(* Create Drive State Output *)
CASE DriveMode OF
0:
	IF bModePMActive THEN
		(* Parameterization mode active *)
		DriveState := DriveState_Mode_PM;
	ELSE
		(* Mode Invalid *)
		DriveState := DriveState_Mode_Invalid;
	END_IF
1:
	IF bModePMActive THEN
		(* Mode Invalid *)
		DriveState := DriveState_Mode_Invalid;
	ELSE
		(* 'bb' mode active *)
		DriveState := DriveState_Mode_bb;
	END_IF
2:
	IF bModePMActive THEN
		(* Mode Invalid *)
		DriveState := DriveState_Mode_Invalid;
	ELSE
		(* Ab' mode active *)
		DriveState := DriveState_Mode_Ab;
	END_IF
3:
	IF bModePMActive THEN
		(* Mode Invalid *)
		DriveState := DriveState_Mode_Invalid;
	ELSE
		IF bDriveHalt THEN
			(* 'AH' mode active *)
			DriveState := DriveState_Mode_AH;
		ELSE
			IF NOT bMLDRunning THEN
				(* 'AF' mode active *)
				DriveState := DriveState_Mode_AF;
			ELSE
				IF bPressureControlActive THEN
					(* Pressure control mode active *)
					DriveState := DriveState_Mode_PC;
				ELSE
					(* flow rate control mode active *)
					DriveState := DriveState_Mode_FC;
				END_IF
			END_IF
		END_IF
	END_IF
ELSE
	(* Mode Invalid *)
	DriveState := DriveState_Mode_Invalid;
END_CASE

(* Mode specific operations and calculations *)
CASE DriveState OF

DriveState_Mode_PC:
(* Pressure Control Mode Active *)
	CommandValueReached := bPressureCmdValReached;
	(* start Pump01 if commanded *)
	Pump01On := PumpOn;

	(* Pump02 is controlled from MLD program *)
	Pump02On := PumpOn AND bMLDPump2OnCmd;

	(* initialize total volume *)
	IF Pump01On THEN
		dwTotalVolume := VolumePump01;
		IF Pump02On THEN
			dwTotalVolume := VolumePump01 + VolumePump02;
		END_IF
	ELSE
		dwTotalVolume := 0;
	END_IF
	(* flow rate is multiplication of Act Velocity and total volume *)
	FlowrateActValue := dwTotalVolume * diVelocityAct ;
	(* transfer Pressure Command value to drive *)
	diPressureCmd := PressureCmdValue;
	(* reset velocty command *)
	diVelocityCmd := 0;

DriveState_Mode_FC:
(* Flow rate Control Mode Active *)
	(* Flow rate value reached when Velocity is within tolerance window *)
	CommandValueReached := bVelCmdValReached;
	(* start Pump01 if commanded *)
	Pump01On := PumpOn;
	(* Pump02 is on along with Pump01 *)
	Pump02On := PumpOn ;

	(* initialize total volume *)
	IF Pump01On THEN (* and Pump02 is also On *)
		dwTotalVolume := VolumePump01 + VolumePump02;
	ELSE
		dwTotalVolume := 0;
	END_IF
	(* flow rate is multiplication of Act Velocity and total volume *)
	FlowrateActValue := dwTotalVolume * diVelocityAct ;

	IF (dwTotalVolume = 0 ) THEN
		(* reset velocty command, no Volume no flow rate control *)
		diVelocityCmd := 0;
	ELSE
		(* velocty command value is derived by deviding Flowrate Command value with Total volume *)
		diVelocityCmd := FlowrateCmdValue / dwTotalVolume;
	END_IF

	(* Pressure Command zero in Flow rate control *)
	diPressureCmd := 0;
ELSE
	(* reset all outputs if not in Process Control mode *)
	dwTotalVolume := 0;
	diVelocityCmd := 0;
	FlowrateActValue := 0;
	diPressureCmd := 0;
	CommandValueReached := FALSE;
END_CASE
(* end of Mode specific operations *)

(* set Master control word and Signal control word *)
wMasterControlWord.14 := DriveEnable;
wMasterControlWord.15 := DriveStart;
wMasterControlWord.13 := DriveStart;                                       (* Drive Halt bit must be set to Activate AF mode at Drive*)

(* reset Diagnostic message using Signal control Word Bit 5 , S144 *)
wSignalControlWord.5 := ResetDriveError;

(* Command for changing the operating mode from Pressure control to Flow rate control and vice versa *)
IF ( OperatingMode = 1)  AND DriveEnable AND DriveStart THEN
	wMLDControlWord.0 := TRUE;
ELSE
	wMLDControlWord.0 := FALSE;
END_IF
(* command to open / close Pump 01 *)
wMLDControlWord.2 := Pump01On;

(* Transfer Command values to the respective output variables *)
stOutputPara.wMasterControlWord := wMasterControlWord;
fbMuxIndradrive.dwValue_WRITE_2 := WORD_TO_DWORD(wSignalControlWord);
fbMuxIndradrive.dwValue_WRITE_3 := diVelocityCmd;
fbMuxIndradrive.dwValue_WRITE_4 := diPressureCmd;
fbMuxIndradrive.dwValue_WRITE_5 := WORD_TO_DWORD (wMLDControlWord);

(*###############################################################################*)
(*####  Call Multiplex Function block and get element number '0' Read and Written Cyclically                      *)
(*###############################################################################*)
fbMuxIndradrive(
	uiINDEX_WRITE                          := OP_MODE_PROCESS_CNTRL ,
	uiLIST_INDEX_WRITE                := LIST_INDEX_0,
	dwValue_WRITE_1                     :=  ,       (* S-0-0000 - Reserve *)
	dwValue_WRITE_2                     :=  ,       (* S-0-0145 - Signal control word *)
	dwValue_WRITE_3                     :=  ,       (* S-0-0259 - Positioning Velocity*)
	dwValue_WRITE_4                     :=  ,       (* S-0-0282 - Position Command Value *)
	dwValue_WRITE_5                     :=  ,       (* S-0-0000 - Reserve *)
	dwValue_WRITE_6                     :=  ,       (* S-0-0000 - Reserve *)
	dwValue_WRITE_7                     :=  ,       (* S-0-0000 - Reserve *)
	dwValue_WRITE_8                     :=  ,       (* S-0-0000 - Reserve *)
	uiINDEX_READ                           := OP_MODE_PROCESS_CNTRL,
	uiLIST_INDEX_READ                 := LIST_INDEX_0 ,
	stEK_IN                                         := stInputPara.stMUX_in ,
	uiINDEX_WRITE_ACKNOWLEDGE=> ,
	uiLIST_INDEX_WRITE_ACKNOWLEDGE=> ,
	uiINDEX_READ_ACKNOWLEDGE=> ,
	uiLIST_INDEX_READ_ACKNOWLEDGE=> ,
	dwValue_READ_1                      => ,           (* S-0-0000 - Reserve *)
	dwValue_READ_2                      => ,           (* S-0-0144 - Signal Status word *)
	dwValue_READ_3                      => ,           (* S-0-0047 - Velocity feedback value *)
	dwValue_READ_4                      => ,           (* S-0-0051 - Postion feedback value *)
	dwValue_READ_5                      => ,           (* S-0-0390 - Drive Diagnostic word *)
	dwValue_READ_6                      => ,           (* S-0-0000 - Reserve *)
	dwValue_READ_7                      => ,           (* S-0-0000 - Reserve *)
	dwValue_READ_8                      => ,           (* S-0-0000 - Reserve *)
	stEK_OUT                                    => stOutputPara.stMUX_out);
END_FUNCTION_BLOCK

(* POU fbIndradrive, ST *)
FUNCTION_BLOCK fbIndradrive
VAR_INPUT
	In_Enable:BOOL;			(*1=Enable Drive, 0=Disable and ignore error*)
	In_Reset:BOOL;
	In_AbsEncoder:BOOL;		(*1=Absolute Encoder, 0=Incremental Encoder*)
	In_DriveInput:st_Indradrive_DCP_input ;		(*Indradrive Input Words via Ethercat*)
	In_CommState:UINT ;		(*Ethercat Slave State, 8=OK*)
	plsResetMode: R_TRIG;
END_VAR
VAR_OUTPUT
	Out_DriveOutput: st_Indradrive_DCP_output;	(*Indradrive Output Words via Ethercat*)
	Out_DriveFeedRateOverride: UINT;			(*Indradrive Output for Feedrate override, keep at 100%*)
END_VAR
VAR_IN_OUT
	DriveVar:structIndradrive;	(*Local Data structure to handle Indradrive variables*)
	Station:Struc_Station_Ctrl ;
END_VAR
VAR
	Drive: FB_Indradrive_DCP;	(*Standard Function Block Provided by Bosch*)
	tmrDriveEnableTOUT:TON;
	tmrHomingTOUT:TON;
	tmrMovePosTOUT:TON;
	diPosCmd:DINT;
	diVelCmd:DINT;
	DriveStatus:INT;
	plsInPos: R_TRIG;
	plsLimitTriggered: R_trig;
	plsMoveRel: R_trig;
	plsStopMove: R_TRIG;
	plsEMGReset: R_trig;
	ServoBusy:BOOL;
	NotAbsEncHoming:BOOL;
	plsMoveAbs: R_trig;
	plsStopMove2: R_trig;
END_VAR
VAR CONSTANT
	FACTOR_DINT_REAL : INT := 10000;
	FACTOR_VEL_DINT_REAL : INT := 1000;
END_VAR
(* convert DINT values from FB to REAL values for the user program and vise versa*)
(* used only for trace purpose *)
DriveVar.Out_CurrPos := DINT_TO_REAL(Drive.diPOS_ACT) / FACTOR_DINT_REAL;
DriveVar.Out_CurrVel := DINT_TO_REAL(Drive.diVEL_ACT) / FACTOR_VEL_DINT_REAL;

(* REAL variables can be used for commanding instead of DINT variable used in the sample code *)
Drive.diPOS_CMD := REAL_TO_DINT (DriveVar.In_PosCmd * FACTOR_DINT_REAL);
Drive.diVEL_CMD := REAL_TO_DINT (DriveVar.In_VelCmd * FACTOR_VEL_DINT_REAL);

(*Force Slow Speed in Manual Mode When close to Negative Limit For Accurate Referencing*)
IF DriveVar.Out_CurrPos <= 20 AND DriveVar.In_JogBwd THEN
	Drive.diVEL_CMD := 60 * FACTOR_VEL_DINT_REAL;
END_IF

IF mc.ManualMode AND DriveVar.In_VelCmd > 1000 THEN
	DriveVar.In_VelCmd := 1000;
END_IF

Out_DriveFeedRateOverride := 100;

(***********************************************************************************************)
(*Servo Controller Status*)

IF NOT In_DriveInput.wSignalstatuswort.11 AND NOT In_DriveInput.wSignalstatuswort.12 THEN
	DriveStatus := 0;	(* Control section and power section not ready for operation (e.g., drive error or phase 2)*)
ELSIF NOT In_DriveInput.wSignalstatuswort.11 AND In_DriveInput.wSignalstatuswort.12 THEN
	DriveStatus := 1;	(* Control section ready for operation (bb)*)
ELSIF In_DriveInput.wSignalstatuswort.11 AND NOT In_DriveInput.wSignalstatuswort.12 THEN
	DriveStatus := 2;	(* Control section and power section ready for operation (Ab)*)
ELSIF In_DriveInput.wSignalstatuswort.11 AND In_DriveInput.wSignalstatuswort.12 THEN
	DriveStatus := 3;	(* Drive with torque (AF)*)
END_IF

(***********************************************************************************************)
(*Servo Limit Sensors Status*)
DriveVar.Out_PosLimit := In_DriveInput.wSignalstatuswort.13;
DriveVar.Out_NegLimit := In_DriveInput.wSignalstatuswort.14;

(***********************************************************************************************)
(*Error Handling*)

IF In_Reset THEN
	DriveVar.Out_ErrorWord := 0;
END_IF

Drive.bRESET := In_Reset;

(*Servo is in Alarm State Error*)
IF Drive.bERROR AND In_Enable  THEN
	DriveVar.Out_ErrorWord := 11;
END_IF

(*Servo Control and Power Section Not Ready Error*) 
IF DriveStatus = 0 AND In_Enable  THEN
	DriveVar.Out_ErrorWord := 12;
END_IF

(*Servo Enable Timeout Error*) 
tmrDriveEnableTOUT(IN:= Drive.bDRIVE_ENABLE AND NOT (Drive.bQ_DRIVE_ENABLE ),PT:=T#5S);
IF tmrDriveEnableTOUT.Q AND In_Enable THEN
	DriveVar.Out_ErrorWord := 13;
END_IF

(*Servo Not Referenced Error*)
IF Drive.bQ_DRIVE_ENABLE AND NOT Drive.bIN_REFERENCE AND In_AbsEncoder AND In_Enable  THEN
	DriveVar.Out_ErrorWord := 20;
END_IF

(*Servo Homing Timeout Error*) 
tmrHomingTOUT(IN:= Drive.bHOMING,PT:=T#3000S);
IF tmrHomingTOUT.Q THEN 
	DriveVar.Out_ErrorWord := 21;
	Drive.bHOMING := FALSE;
END_IF

(*Servo Move Position Timeout Error*) 
tmrMovePosTOUT(IN:= (DriveVar.In_MoveAbs OR ServoBusy OR
					DriveVar.In_MoveRel) AND NOT DriveVar.Out_InPos,PT:=T#300S);
IF tmrMovePosTOUT.Q THEN 
	DriveVar.Out_ErrorWord := 22;
	ServoBusy := FALSE;
	DriveVar.In_MoveAbs := FALSE;
	DriveVar.In_MoveRel := FALSE;
END_IF

(*Servo Move Position Limit Error*) 
IF ServoBusy AND
	(((DriveVar.In_PosCmd < DriveVar.Out_CurrPos) AND NOT DriveVar.Out_NegLimit) 
	OR ((DriveVar.In_PosCmd > DriveVar.Out_CurrPos) AND NOT DriveVar.Out_PosLimit)) THEN 
	DriveVar.Out_ErrorWord := 23;
	ServoBusy := FALSE;
	DriveVar.In_MoveAbs := FALSE;
	DriveVar.In_MoveRel := FALSE;
END_IF

(*Servo Communication Error*) 
IF In_CommState <> 8 AND In_Enable  THEN
	DriveVar.Out_ErrorWord := 10;
END_IF

IF DriveVar.Out_ErrorWord > 1 THEN
	DriveVar.Out_Error := TRUE;
ELSE
	IF NOT DriveVar.In_MoveXLock THEN
		DriveVar.Out_ErrorWord := 0;
	ELSE
		DriveVar.Out_ErrorWord := 1;
	END_IF
	DriveVar.Out_Error := FALSE;
END_IF
(*Warning*)
DriveVar.Out_Warning := Drive.bWARNING;

(***********************************************************************************************)
(*Servo Enable*)

plsLimitTriggered(CLK:=NOT (DriveVar.Out_NegLimit AND DriveVar.Out_PosLimit) AND NOT NotAbsEncHoming);

IF plsLimitTriggered.Q THEN
	DriveVar.In_ServoOn		 := FALSE;
END_IF

IF In_Enable AND DriveVar.In_ServoOn AND NOT DriveVar.Out_Error
	AND DriveStatus >= 1  THEN
	(* drive enable and drive on commands *)
	Drive.bDRIVE_ENABLE	:= TRUE;
	Drive.bDRIVE_START		:= TRUE;
ELSE
	(* drive enable and drive on commands *)
	Drive.bDRIVE_ENABLE	:= FALSE;
	Drive.bDRIVE_START		:= FALSE;
	DriveVar.Out_Busy 		:= FALSE;
	DriveVar.In_JogBwd 		:= FALSE;
	DriveVar.In_JogFwd 		:= FALSE;
	DriveVar.In_MoveAbs 		:= FALSE;
	DriveVar.In_MoveHome 	:= FALSE;
	DriveVar.In_MoveRel 		:= FALSE;
	DriveVar.In_ServoOn 		:= FALSE;
END_IF

Drive.bIMMEDIATE_CHANGE := TRUE;
	
(***********************************************************************************************)
(*Servo Movement Control*)
(***********************************************************************************************)

(*Force Stop Command When Mode Changes*)
plsResetMode(CLK:= NOT MC.AutoMode);

plsStopMove(CLK:= NOT (Station.OriginSchRun OR MC.OriginSchRun OR
						Station.AutoRun OR Station.M_Step));

plsStopMove2(CLK:= (Station.OriginSchRun OR MC.OriginSchRun OR
						Station.M_Step OR MC.AutoMode));
						
IF plsStopMove.Q AND plsStopMove2.Q OR plsResetMode.Q THEN
	DriveVar.In_StopMove := TRUE;
	DriveVar.In_MoveAbs := FALSE;
	DriveVar.In_MoveHome := FALSE;
	DriveVar.In_MoveRel := FALSE;
END_IF

(*Check New Move Command Direction for Interlocking Purpose*)
IF DriveVar.In_JogFwd OR 
	((DriveVar.In_PosCmd > DriveVar.Out_CurrPos) AND
		DriveVar.In_MoveAbs) OR
	((DriveVar.In_PosCmd > 0) AND
		DriveVar.In_MoveRel) THEN
	DriveVar.Out_PosDirc := TRUE;
	DriveVar.Out_NegDirc := FALSE;
ELSIF DriveVar.In_JogBwd OR 
	((DriveVar.In_PosCmd < DriveVar.Out_CurrPos) AND
		DriveVar.In_MoveAbs) OR
	((DriveVar.In_PosCmd < 0) AND
		DriveVar.In_MoveRel) THEN	
	DriveVar.Out_PosDirc := FALSE;
	DriveVar.Out_NegDirc := TRUE;
ELSE
	DriveVar.Out_PosDirc := FALSE;
	DriveVar.Out_NegDirc := FALSE;
END_IF


(* Origin Search for Incremental Encoder Servo*)
	IF NOT In_AbsEncoder THEN
		IF Drive.bIN_REFERENCE OR NOT DriveVar.In_ServoOn THEN
			Drive.bHOMING 		:= FALSE;
			NotAbsEncHoming	:=FALSE;
		END_IF

		IF DriveVar.In_MoveHome  AND
			Drive.bQ_DRIVE_ENABLE AND
			DriveStatus = 3  AND
			NOT DriveVar.Out_Busy THEN
			Drive.bHOMING 		:= TRUE;
			NotAbsEncHoming	:=TRUE;
		END_IF
	END_IF

IF Drive.bQ_DRIVE_ENABLE AND Drive.bQ_MAIN_MODE AND DriveStatus = 3 THEN
	DriveVar.Out_Ready := TRUE;
	


	(*Jog Command*)
	IF MC.ManualMode AND NOT Station.M_Step THEN
		IF DriveVar.In_JogFwd AND NOT DriveVar.In_JogBwd AND DriveVar.In_MoveXLock THEN
			(* Jog Positive command *)
			Drive.bJOG_FORWARD := TRUE;
			Drive.bJOG_BACKWARD := FALSE;
		ELSIF NOT DriveVar.In_JogFwd AND DriveVar.In_JogBwd AND DriveVar.In_MoveXLock THEN
			(* Jog Negative  command *)
			Drive.bJOG_FORWARD := FALSE;
			Drive.bJOG_BACKWARD := TRUE;
		ELSE
			(* Stop Jogging *)
			Drive.bJOG_FORWARD := FALSE;
			Drive.bJOG_BACKWARD := FALSE;
		END_IF
	ELSE
		DriveVar.In_JogFwd := FALSE;
		DriveVar.In_JogBwd := FALSE;
	END_IF
	
	IF Drive.bIN_REFERENCE THEN
		IF DriveVar.In_MoveXLock THEN
			(* Start Absolute move *)
			plsMoveAbs(CLK:=DriveVar.In_MoveAbs);
			IF DriveVar.In_MoveAbs AND Drive.bNEW_VALUE_POSSIBLE THEN
				ServoBusy := TRUE;
				(*DriveVar.In_MoveAbs := FALSE;*)
				IF Drive.diPOS_CMD <> Drive.diPOS_ACT AND Drive.diVEL_CMD <> 0 THEN
					DriveVar.Out_InPos := FALSE;
					Drive.bABS_REL := FALSE;       				(* False --> Absolute command *)
					IF Drive.bNEW_VALUE THEN
						Drive.bNEW_VALUE := FALSE;
					ELSE
						Drive.bNEW_VALUE := TRUE;
					END_IF
				END_IF
			END_IF
			(* Start Relative move *)
			plsMoveRel(CLK:=DriveVar.In_MoveRel);
			IF plsMoveRel.Q AND Drive.bNEW_VALUE_POSSIBLE AND 
				NOT ServoBusy  THEN
				ServoBusy := TRUE;
				DriveVar.In_MoveRel := FALSE;
				IF Drive.diPOS_CMD <> 0 AND Drive.diVEL_CMD <> 0 THEN
					DriveVar.Out_InPos := FALSE;
					Drive.bABS_REL := TRUE;       				(* True  --> Relative  command *)
					IF Drive.bNEW_VALUE THEN
						Drive.bNEW_VALUE := FALSE;
					ELSE
						Drive.bNEW_VALUE := TRUE;
					END_IF
				END_IF
			END_IF
		END_IF
	ELSE
		DriveVar.Out_InPos := FALSE;
	END_IF
	
	(*Set Servo Busy Status*)	
	DriveVar.Out_Busy := NOT Drive.bIN_STANDSTILL;
	IF DriveVar.Out_Busy THEN
		DriveVar.Out_InPos := FALSE; 
	END_IF
	
ELSE

	ServoBusy 				:= FALSE;
	DriveVar.In_MoveAbs 		:= FALSE;
	DriveVar.In_MoveRel		 := FALSE;
	DriveVar.Out_Ready		:= FALSE;
	DriveVar.In_JogBwd		 := FALSE;
	DriveVar.In_JogFwd 		:= FALSE;
(*	DriveVar.In_MoveHome 	:= FALSE;*)
	Drive.bJOG_FORWARD	:= FALSE;
	Drive.bJOG_BACKWARD	 := FALSE;
	Drive.bHOMING			 := FALSE;

END_IF

(* wait for InPos *)
plsInPos(CLK:= Drive.bPOS_OK);
plsEMGReset(CLK:= NOT MC.Trouble );
IF Drive.bPOS_OK AND 
	fcComparePos(CurrPos:= DriveVar.In_PosCmd, TargetPos:= DriveVar.Out_CurrPos,Tolerance:=0.5)
	AND Drive.bIN_STANDSTILL AND Drive.bNEW_VALUE_POSSIBLE  THEN
	DriveVar.Out_InPos 		:= TRUE;
	DriveVar.In_MoveAbs 		:= FALSE;
	DriveVar.In_MoveRel		:= FALSE;
	ServoBusy 				:= FALSE;
END_IF

IF plsEMGReset.Q AND Drive.bIN_STANDSTILL AND Drive.bIN_REFERENCE AND
	Drive.bNEW_VALUE_POSSIBLE THEN
	DriveVar.Out_InPos		:= TRUE;
	ServoBusy 				:= FALSE;
END_IF

IF DriveVar.In_StopMove THEN
	DriveVar.In_MoveAbs 		:= FALSE;
	DriveVar.In_MoveHome	:= FALSE;
	DriveVar.In_MoveRel		:= FALSE;
	DriveVar.In_JogBwd 		:= FALSE;
	DriveVar.In_JogFwd		:= FALSE;
	DriveVar.In_StopMove 		:= FALSE;
	(* Stop Movement *)
	Drive.bJOG_FORWARD	:= TRUE;
	Drive.bJOG_BACKWARD 	:= TRUE;
	ServoBusy 				:= FALSE;

ELSIF 	Drive.bJOG_FORWARD AND Drive.bJOG_BACKWARD AND MC.AutoMode THEN
	Drive.bJOG_FORWARD 	:= FALSE;
	Drive.bJOG_BACKWARD 	:= FALSE;
END_IF


(***********************************************************************************************)
(*Servo Function Block*)


Drive(
	bJOG_FORWARD:= 			,
	bJOG_BACKWARD:=			,
	bNEW_VALUE:= ,
	bABS_REL:= ,
	bIMMEDIATE_CHANGE:= ,
	diPOS_CMD:= ,
	diVEL_CMD:= , 
	stEK_IN:=					In_DriveInput ,
	bQ_DRIVE_ENABLE=> ,
	bQ_MAIN_MODE=> , 
	bIN_REFERENCE=> , 
	bPOS_OK=> , 
	bNEW_VALUE_POSSIBLE=> , 
	bSTATUS_MESSAGE=> , 
	bWARNING=> , 
	bERROR=> , 
	bIN_STANDSTILL=> , 
	dwDRIVE_DIAGNOSIS=> , 
	diPOS_ACT=> , 
	diVEL_ACT=> ,
	stEK_OUT=>					Out_DriveOutput );


	Out_DriveOutput.wSignalsteuerwort.6 	:= drive.bJOG_FORWARD;
	Out_DriveOutput.wSignalsteuerwort.7 	:= drive.bJOG_BACKWARD;
	Out_DriveOutput.wSignalsteuerwort.15 :=  NotAbsEncHoming  ;

	
(***********************************************************************************************)
(*Set Reference Point for Absulute Encoder Servo*)
	Out_DriveOutput.wSignalsteuerwort.1 := DriveVar.In_SetAbsRef;
	DriveVar.Out_Referenced := Drive.bIN_REFERENCE;
END_FUNCTION_BLOCK

(* POU fcComparePos, ST *)
FUNCTION fcComparePos : BOOL
VAR_INPUT
	CurrPos		:REAL;
	TargetPos	:REAL;
	Tolerance	:REAL;
END_VAR
VAR
END_VAR
IF 	CurrPos >= 	(TargetPos	-	Tolerance) AND
	CurrPos <= 	(TargetPos	+	Tolerance) THEN
	fcComparePos := TRUE;
ELSE
	fcComparePos := FALSE;
END_IF
END_FUNCTION

(* POU Std_Cylinder_Ctrl, LD *)
FUNCTION_BLOCK Std_Cylinder_Ctrl

VAR_INPUT
	IN:BOOL;
	IN_CylName:STRING;
	In_Enable:BOOL;
	In_Reset:BOOL;


	(*Trigger*)
	In_AutoWork:BOOL;
	In_AutoHome:BOOL;
	In_OrgWork:BOOL;
	In_OrgHome:BOOL;
	(*Mechanical Interlock*)
	In_WorkXLock:BOOL;
	In_HomeXLock:BOOL;
	(*Sensors*)
	In_WorkRS:BOOL;
	In_HomeRS:BOOL;

	(*Timer*)
	In_WorkTON:TIME;
	In_HomeTON:TIME;
	in_Timeout:TIME;
END_VAR

VAR_OUTPUT
	Q:BOOL;
	Out_WorkSV:BOOL;
	Out_HomeSV:BOOL;
	E_WorkErr:BOOL;
	E_HomeErr:BOOL;
	S_WorkPos:BOOL;
	S_HomePos:BOOL;
END_VAR

VAR
	(* Trigger*)
	T_ManWork:BOOL;
	T_ManHome:BOOL;

	Loc_Work:BOOL;
	Loc_Home:BOOL;
	Err_Cyl:BOOL;
	Fwd_TOut: TON;
	Bwd_TOut: TON;
	Fwd_TON: TON;
	Bwd_TON: TON;
	Loc_WorkPls: BOOL;
	FwdPls: R_TRIG;
	BwdPls: R_TRIG;
	Loc_HomePls: BOOL;
	Out_RSErr:BOOL;
	FwdPosPls: F_TRIG;
	BwdPosPls: F_TRIG;
END_VAR
VAR_IN_OUT

END_VAR
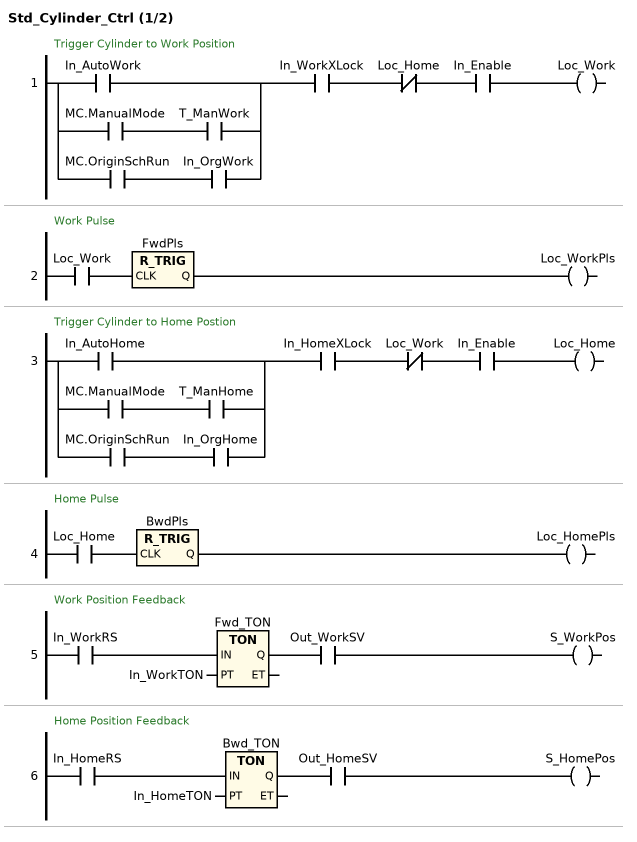
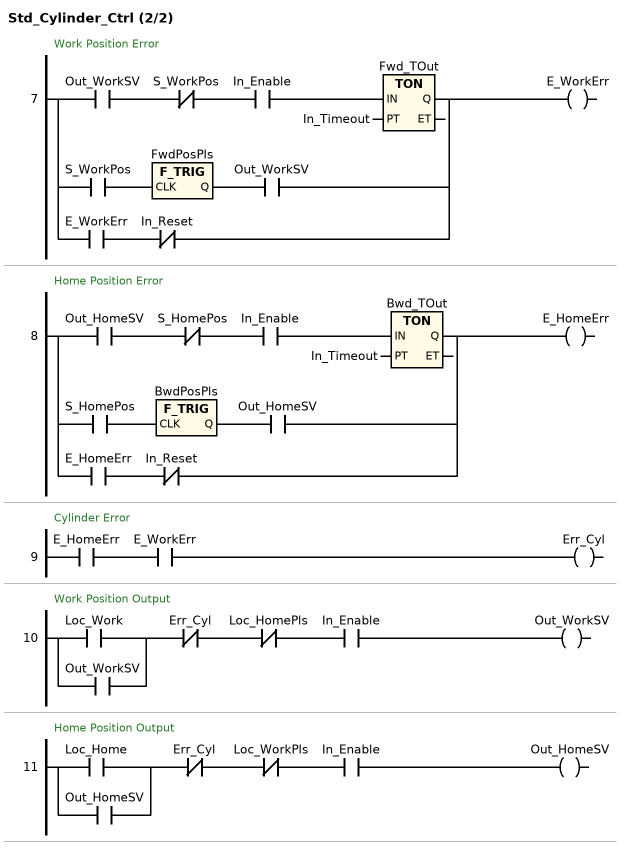
_LD_ (* Ladder Diagram *)
NETWORK 1 (* Trigger Cylinder to Work Position *)
	{ [In_AutoWork] | [MC.ManualMode] - [T_ManWork] | [MC.OriginSchRun] - [In_OrgWork] } - [In_WorkXLock] - [/Loc_Home] - [In_Enable] --- (Loc_Work)
NETWORK 2 (* Work Pulse *)
	[Loc_Work] - FwdPls:R_TRIG(CLK: *) --- (Loc_WorkPls)
NETWORK 3 (* Trigger Cylinder to Home Postion *)
	{ [In_AutoHome] | [MC.ManualMode] - [T_ManHome] | [MC.OriginSchRun] - [In_OrgHome] } - [In_HomeXLock] - [/Loc_Work] - [In_Enable] --- (Loc_Home)
NETWORK 4 (* Home Pulse *)
	[Loc_Home] - BwdPls:R_TRIG(CLK: *) --- (Loc_HomePls)
NETWORK 5 (* Work Position Feedback *)
	[In_WorkRS] - Fwd_TON:TON(IN: *, PT: In_WorkTON) - [Out_WorkSV] --- (S_WorkPos)
NETWORK 6 (* Home Position Feedback *)
	[In_HomeRS] - Bwd_TON:TON(IN: *, PT: In_HomeTON) - [Out_HomeSV] --- (S_HomePos)
NETWORK 7 (* Work Position Error *)
	{ [Out_WorkSV] - [/S_WorkPos] - [In_Enable] - Fwd_TOut:TON(IN: *, PT: In_Timeout) | [S_WorkPos] - FwdPosPls:F_TRIG(CLK: *) - [Out_WorkSV] | [E_WorkErr] - [/In_Reset] } --- (E_WorkErr)
NETWORK 8 (* Home Position Error *)
	{ [Out_HomeSV] - [/S_HomePos] - [In_Enable] - Bwd_TOut:TON(IN: *, PT: In_Timeout) | [S_HomePos] - BwdPosPls:F_TRIG(CLK: *) - [Out_HomeSV] | [E_HomeErr] - [/In_Reset] } --- (E_HomeErr)
NETWORK 9 (* Cylinder Error *)
	[E_HomeErr] - [E_WorkErr] --- (Err_Cyl)
NETWORK 10 (* Work Position Output *)
	{ [Loc_Work] | [Out_WorkSV] } - [/Err_Cyl] - [/Loc_HomePls] - [In_Enable] --- (Out_WorkSV)
NETWORK 11 (* Home Position Output *)
	{ [Loc_Home] | [Out_HomeSV] } - [/Err_Cyl] - [/Loc_WorkPls] - [In_Enable] --- (Out_HomeSV)
_END_LD_
(* the same logic as Structured Text *)
(* Network 1: Trigger Cylinder to Work Position *)
Loc_Work := (In_AutoWork OR MC.ManualMode AND T_ManWork OR MC.OriginSchRun AND In_OrgWork) AND In_WorkXLock AND NOT Loc_Home AND In_Enable;
(* Network 2: Work Pulse *)
FwdPls(CLK := Loc_Work);
Loc_WorkPls := FwdPls.Q;
(* Network 3: Trigger Cylinder to Home Postion *)
Loc_Home := (In_AutoHome OR MC.ManualMode AND T_ManHome OR MC.OriginSchRun AND In_OrgHome) AND In_HomeXLock AND NOT Loc_Work AND In_Enable;
(* Network 4: Home Pulse *)
BwdPls(CLK := Loc_Home);
Loc_HomePls := BwdPls.Q;
(* Network 5: Work Position Feedback *)
Fwd_TON(IN := In_WorkRS, PT := In_WorkTON);
S_WorkPos := Fwd_TON.Q AND Out_WorkSV;
(* Network 6: Home Position Feedback *)
Bwd_TON(IN := In_HomeRS, PT := In_HomeTON);
S_HomePos := Bwd_TON.Q AND Out_HomeSV;
(* Network 7: Work Position Error *)
Fwd_TOut(IN := Out_WorkSV AND NOT S_WorkPos AND In_Enable, PT := In_Timeout);
FwdPosPls(CLK := S_WorkPos);
E_WorkErr := Fwd_TOut.Q OR FwdPosPls.Q AND Out_WorkSV OR E_WorkErr AND NOT In_Reset;
(* Network 8: Home Position Error *)
Bwd_TOut(IN := Out_HomeSV AND NOT S_HomePos AND In_Enable, PT := In_Timeout);
BwdPosPls(CLK := S_HomePos);
E_HomeErr := Bwd_TOut.Q OR BwdPosPls.Q AND Out_HomeSV OR E_HomeErr AND NOT In_Reset;
(* Network 9: Cylinder Error *)
Err_Cyl := E_HomeErr AND E_WorkErr;
(* Network 10: Work Position Output *)
Out_WorkSV := (Loc_Work OR Out_WorkSV) AND NOT Err_Cyl AND NOT Loc_HomePls AND In_Enable;
(* Network 11: Home Position Output *)
Out_HomeSV := (Loc_Home OR Out_HomeSV) AND NOT Err_Cyl AND NOT Loc_WorkPls AND In_Enable;
END_FUNCTION_BLOCK

(* POU Std_Hist_StepCase, ST *)
FUNCTION_BLOCK Std_Hist_StepCase

VAR_INPUT
	IN:BOOL;
	CurrentStep:INT;
	NextStep:INT;
END_VAR

VAR_OUTPUT
	Q:BOOL;
	NewStep:INT;
END_VAR

VAR
	StepData:ARRAY[0..100] OF Struc_Hist_Step_Case ;

	StepTimer: TON;
	Loop: INT;
END_VAR
IF CurrentStep = NextStep THEN
StepTimer(IN:=TRUE , PT:=t#1100h , Q=> , ET=> );

StepData[0].CurrentStepHist :=CurrentStep;

ELSE
(* Copy HIstory File *)
FOR Loop := 0 TO 99 DO
StepData[100-Loop].CurrentStepHist   := StepData[99-Loop].CurrentStepHist ;
StepData[100-Loop].NextStepHist := StepData[99-Loop].NextStepHist ;
StepData[100-Loop].StepTime := StepData[99-Loop].StepTime;
END_FOR

(* Update New Data*)
StepData[1].NextStepHist:=NextStep;
StepData[1].StepTime :=StepTimer.ET;

StepTimer(IN:=FALSE , PT:=T#1100h , Q=> , ET=> );
NewStep:=NextStep;
END_IF
END_FUNCTION_BLOCK

(* POU Std_IAI_16Point, ST *)
(* @OBJECTFLAGS := '0, 8' *)
FUNCTION_BLOCK Std_IAI_16Point
VAR_INPUT
	In_Enable:BOOL;
	In_Name:STRING;
	In_AutoMode:BOOL;

	(*Trigger*)
	In_AutoStart:BOOL;
	In_OrgHome:BOOL;

	In_Pos_Num:WORD;
	In_ALM:BOOL;
	In_Reset:BOOL;
	In_PEND:BOOL;
	In_HEND:BOOL;
	In_Mec_Interlock:BOOL;
	In_PosTON:TIME;
	In_Timeout:TIME;
END_VAR

VAR_OUTPUT
	S_InPos:BOOL;  (*Current Pos*)
	S_Pos_Num : INT;
	S_InHome:BOOL;
	Out_CSTR:BOOL;
	Out_PC1:BOOL;
	Out_PC2:BOOL;
	Out_PC4:BOOL;
	Out_PC8:BOOL;
	E_Alm:BOOL;
	E_AlmPos:BOOL;
END_VAR

VAR
	(* Trigger*)
	T_ManStart:BOOL;
	T_ManHome:BOOL;
	T_ManPos_Num:INT;

	CSTR:BOOL; (*Common Start Bit*)
	Home : BOOL;
	Pos_Num:INT;

	TimePos: TON;
	BitPos1: BOOL;
	BitPos2: BOOL;
	BitPos3: BOOL;
	BitPos4: BOOL;
	TimeOut: TON;
	TempBit1: BYTE;
	TempBit2: BYTE;
	TempBit3: BYTE;
	TempBit4: BYTE;
	BytePos: BYTE;
	IAI_TimeOut: BOOL;
	Error_Alm: BOOL;
	DoneTon: BOOL;
	tmrStartDelay: TON;
	StartDelayTon: BOOL;
	plsStart: R_TRIG;
	StartDelayPls: BOOL;
	plsIAIDone: R_TRIG;
	DonePls: BOOL;
	plsHome: R_TRIG;
	HomePls: BOOL;
	HomeSearch: BOOL;
	test: BOOL;
	test1: BOOL;
	tmrStartDelay_1: TON;
	StartDelayTon_1: BOOL;
	IAI_Busy: BOOL;
	test_1: BOOL;
	tmrStartDelay_Home: TON;
	StartDelayTon_Home: BOOL;
	tmrStartDelay_Home_1: TON;
	StartDelayTon_Home_1: BOOL;
END_VAR
(**************************************************************************************************************)
(*Trigger*)
(**************************************************************************************************************)
IF  In_AutoStart OR (MC.ManualMode AND T_ManStart) THEN
CSTR := TRUE;
ELSE
CSTR := FALSE;
END_IF;

IF In_AutoMode THEN
Pos_Num := In_Pos_Num;
ELSE
Pos_Num:=T_ManPos_Num;
END_IF


IF (MC.OriginSchRun AND In_OrgHome) OR (MC.ManualMode AND T_ManHome) THEN
Home := TRUE;
Pos_Num:=0;
ELSE
Home := FALSE;
END_IF;
(**************************************************************************************************************)
(*Reset Error/Warning*)
(**************************************************************************************************************)
IF In_reset AND ( E_AlmPos OR E_Alm OR Error_Alm) THEN
	E_AlmPos :=FALSE;
	E_Alm:= FALSE;
	Error_Alm := FALSE;
END_IF;

(**************************************************************************************************************)
(*System Error*)
(**************************************************************************************************************)
(* Time Out*)
TimeOut (IN := Out_CSTR AND NOT S_InPos AND  In_Mec_Interlock, PT:=In_Timeout);
IAI_TimeOut := TimeOut.Q;

IF IAI_TimeOut AND In_Enable THEN
	E_AlmPos := TRUE;
END_IF;

(* IAI Controller Error*)
IF In_Enable AND In_ALM THEN
	E_Alm := TRUE;
END_IF;

(* IAI System In Error Condition*)
Error_Alm := E_AlmPos OR E_Alm;

IF Error_Alm THEN
	Out_CSTR := FALSE;
	S_InPos := FALSE;
	HomeSearch := FALSE;
	IAI_Busy:= FALSE;
END_IF;

(**************************************************************************************************************)
(*Moving To Target Position*)
(**************************************************************************************************************)

Out_PC1 := FALSE;
Out_PC2 := FALSE;
Out_PC4 := FALSE;
Out_PC8 := FALSE;

IF In_Enable AND NOT Error_Alm THEN
	BytePos := INT_TO_BYTE (Pos_Num);
	TempBit1 := BytePos AND 2#1;
	TempBit2 := BytePos AND 2#10;
	TempBit3 := BytePos AND 2#100;
	TempBit4 := BytePos AND 2#1000;

	BitPos1 := INT_TO_BOOL (TempBit1);
	BitPos2 := INT_TO_BOOL (TempBit2);
	BitPos3 := INT_TO_BOOL (TempBit3);
	BitPos4 := INT_TO_BOOL (TempBit4);

		IF BitPos1 THEN
			Out_PC1 := TRUE;
		END_IF;

		IF BitPos2 THEN
			Out_PC2 := TRUE;
		END_IF;

		IF BitPos3 THEN
			Out_PC4 := TRUE;
		END_IF;

		IF BitPos4 THEN
			Out_PC8 := TRUE;
		END_IF;
END_IF;

(**************************************************************************************************************)
(*Moving To Target Position Common*)
(**************************************************************************************************************)
tmrStartDelay(IN := CSTR , PT:= T#0.1s);
StartDelayTon := tmrStartDelay.Q;

plsStart(CLK := StartDelayTon);
StartDelayPls := plsStart.Q;

tmrStartDelay_1(IN := Out_CSTR , PT:= T#0.5s);
StartDelayTon_1 := tmrStartDelay_1.Q;

IF In_Enable AND NOT HomeSearch AND In_Mec_Interlock AND NOT Error_Alm THEN
	IF  StartDelayPls AND In_PEND THEN
		Out_CSTR := TRUE;
		S_InPos := FALSE;
		IAI_Busy := TRUE;
	END_IF;

	IF (StartDelayTon_1 AND Out_CSTR) OR NOT In_PEND  THEN
		Out_CSTR := FALSE;
	END_IF;
END_IF;

(**************************************************************************************************************)
(*Moving Done Complete Status*)
(**************************************************************************************************************)

TimePos (IN :=  In_PEND  AND (IAI_Busy OR HomeSearch) , PT:= In_PosTON);
DoneTon := TimePos.Q;

plsIAIDone(CLK := DoneTon);
DonePls := plsIAIDone.Q;

IF DoneTon AND In_Enable THEN
	IF HomeSearch THEN
		S_Pos_Num := 0;
	ELSE
		S_Pos_Num := Pos_Num;
	END_IF
	S_InPos := TRUE;
	HomeSearch := FALSE;
	IAI_Busy:= FALSE;
END_IF;

(**************************************************************************************************************)
(*Moving Target To Home = Pos 0*)
(**************************************************************************************************************)
S_InHome := S_Pos_Num = 0 AND S_InPos AND In_HEND;

tmrStartDelay_Home(IN := Home   , PT:= T#0.1s);
StartDelayTon_Home := tmrStartDelay_Home.Q;

plsHome (CLK:= StartDelayTon_Home AND NOT IAI_Busy );
HomePls:= plsHome.Q;

tmrStartDelay_Home_1(IN := HomeSearch AND Out_CSTR , PT:= T#0.5s);
StartDelayTon_Home_1 := tmrStartDelay_Home_1.Q;

IF In_Enable AND NOT Error_Alm AND In_Mec_Interlock AND  NOT Out_CSTR  THEN
	IF HomePls THEN
		HomeSearch := TRUE;
		Out_CSTR :=TRUE;
	END_IF;
END_IF;

IF HomeSearch AND StartDelayTon_Home_1 THEN
	Out_CSTR := FALSE;
END_IF;
END_FUNCTION_BLOCK

(* POU Std_IV_Vision_Ctrl, LD *)
FUNCTION_BLOCK Std_IV_Vision_Ctrl
VAR_INPUT
	IN: BOOL;
	In_Name:STRING;
	In_Enable:BOOL;
	In_Alm:BOOL;
	In_Reset:BOOL;
	In_AutoMode:BOOL;
	In_Auto_Model:INT;
	In_Busy:BOOL;
	In_AutoTrigger:BOOL;
	In_Result:BOOL;
	In_Timeout:TIME;
END_VAR

VAR_OUTPUT
	Q:BOOL;
	Out_ProgBit0:BOOL;
	Out_ProgBit1:BOOL;
	Out_ProgBit2:BOOL;
	Out_ProgBit3:BOOL;
	Out_Trigger:BOOL;
	Out_ClearErr:BOOL;
	S_Result:BOOL;
	S_Done:BOOL;
	E_Alm:BOOL;
END_VAR

VAR
	T_ManualTrigger:	BOOL;
	T_Manual_Model:	INT;
	Model:			INT;
	Start:			BOOL;

	TempModel: BYTE;
	ModelBit1: BYTE;
	ModelBit2: BYTE;
	ModelBit3: BYTE;
	ModelBit0: BYTE;
	TimeOut: TON;
	Reset_Result: BOOL;
	Vision_Trigger: R_TRIG;
	tmr_Done: TON;
	Start_Rtrig: R_TRIG;
END_VAR
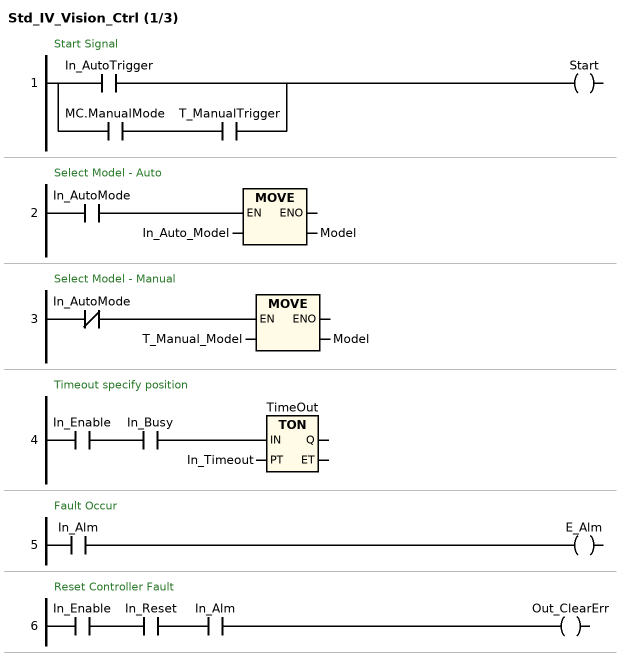
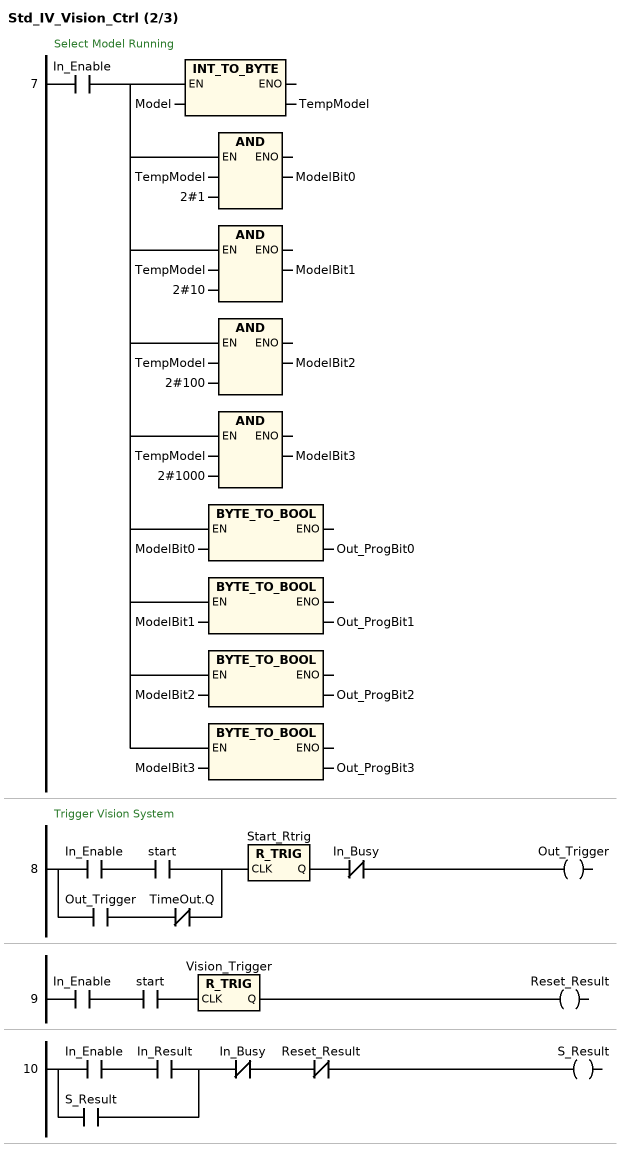
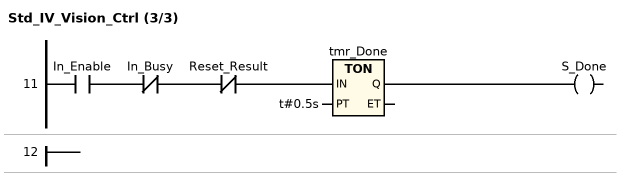
_LD_ (* Ladder Diagram *)
NETWORK 1 (* Start Signal *)
	{ [In_AutoTrigger] | [MC.ManualMode] - [T_ManualTrigger] } --- (Start)
NETWORK 2 (* Select Model - Auto *)
	[In_AutoMode]
		EN --- MOVE(In_Auto_Model) => Model
NETWORK 3 (* Select Model - Manual *)
	[/In_AutoMode]
		EN --- MOVE(T_Manual_Model) => Model
NETWORK 4 (* Timeout specify position *)
	[In_Enable] - [In_Busy] - TimeOut:TON(IN: *, PT: In_Timeout)
NETWORK 5 (* Fault Occur *)
	[In_Alm] --- (E_Alm)
NETWORK 6 (* Reset Controller Fault *)
	[In_Enable] - [In_Reset] - [In_Alm] --- (Out_ClearErr)
NETWORK 7 (* Select Model Running *)
	[In_Enable]
		EN --- INT_TO_BYTE(Model) => TempModel
		EN --- AND(TempModel, 2#1) => ModelBit0
		EN --- AND(TempModel, 2#10) => ModelBit1
		EN --- AND(TempModel, 2#100) => ModelBit2
		EN --- AND(TempModel, 2#1000) => ModelBit3
		EN --- BYTE_TO_BOOL(ModelBit0) => Out_ProgBit0
		EN --- BYTE_TO_BOOL(ModelBit1) => Out_ProgBit1
		EN --- BYTE_TO_BOOL(ModelBit2) => Out_ProgBit2
		EN --- BYTE_TO_BOOL(ModelBit3) => Out_ProgBit3
NETWORK 8 (* Trigger Vision System *)
	{ [In_Enable] - [start] | [Out_Trigger] - [/TimeOut.Q] } - Start_Rtrig:R_TRIG(CLK: *) - [/In_Busy] --- (Out_Trigger)
NETWORK 9
	[In_Enable] - [start] - Vision_Trigger:R_TRIG(CLK: *) --- (Reset_Result)
NETWORK 10
	{ [In_Enable] - [In_Result] | [S_Result] } - [/In_Busy] - [/Reset_Result] --- (S_Result)
NETWORK 11
	[In_Enable] - [/In_Busy] - [/Reset_Result] - tmr_Done:TON(IN: *, PT: t#0.5s) --- (S_Done)
NETWORK 12
	*
_END_LD_
(* the same logic as Structured Text *)
(* Network 1: Start Signal *)
Start := In_AutoTrigger OR MC.ManualMode AND T_ManualTrigger;
(* Network 2: Select Model - Auto *)
IF In_AutoMode THEN
	Model := In_Auto_Model;
END_IF;
(* Network 3: Select Model - Manual *)
IF NOT In_AutoMode THEN
	Model := T_Manual_Model;
END_IF;
(* Network 4: Timeout specify position *)
TimeOut(IN := In_Enable AND In_Busy, PT := In_Timeout);
(* Network 5: Fault Occur *)
E_Alm := In_Alm;
(* Network 6: Reset Controller Fault *)
Out_ClearErr := In_Enable AND In_Reset AND In_Alm;
(* Network 7: Select Model Running *)
IF In_Enable THEN
	TempModel := INT_TO_BYTE(Model);
	ModelBit0 := TempModel AND 2#1;
	ModelBit1 := TempModel AND 2#10;
	ModelBit2 := TempModel AND 2#100;
	ModelBit3 := TempModel AND 2#1000;
	Out_ProgBit0 := BYTE_TO_BOOL(ModelBit0);
	Out_ProgBit1 := BYTE_TO_BOOL(ModelBit1);
	Out_ProgBit2 := BYTE_TO_BOOL(ModelBit2);
	Out_ProgBit3 := BYTE_TO_BOOL(ModelBit3);
END_IF;
(* Network 8: Trigger Vision System *)
Start_Rtrig(CLK := In_Enable AND start OR Out_Trigger AND NOT TimeOut.Q);
Out_Trigger := Start_Rtrig.Q AND NOT In_Busy;
(* Network 9 *)
Vision_Trigger(CLK := In_Enable AND start);
Reset_Result := Vision_Trigger.Q;
(* Network 10 *)
S_Result := (In_Enable AND In_Result OR S_Result) AND NOT In_Busy AND NOT Reset_Result;
(* Network 11 *)
tmr_Done(IN := In_Enable AND NOT In_Busy AND NOT Reset_Result, PT := t#0.5s);
S_Done := tmr_Done.Q;
(* Network 12 *)
END_FUNCTION_BLOCK

(* POU Std_Machine_Ctrl, ST *)
FUNCTION_BLOCK Std_Machine_Ctrl

VAR_INPUT
	In_Start_PB:						BOOL;
	In_Stop_PB:						BOOL;
	In_EmgOK:						BOOL;
	In_Door_Sw: 						BOOL;
	In_Pressure_Sw: 					BOOL;
	In_LightCurtainSafeToCross:		BOOL;
	In_LightCurtainOK: 					BOOL;
	In_OtherTrouble: 					BOOL;
	In_Reset_PB:						BOOL;
	In_Start_Enable:					BOOL;
	In_EndProdWPCleared:			BOOL;
	I_StepFwdPB:					BOOL;
	I_StepBwdPB:					BOOL;

END_VAR

VAR_IN_OUT

END_VAR

VAR_OUTPUT
	Out_RedTower:BOOL;
	Out_YelTower :BOOL;
	Out_GrnTower:BOOL;
	Out_Buzzer:BOOL;

END_VAR

VAR
	Loop: INT;
	LoopStation: INT;
(*************************************************************************************************************************************)
(*Status Bit*)
(*************************************************************************************************************************************)

	AllStationStop:BOOL;

(*************************************************************************************************************************************)
(* HMI Bit*)
(*************************************************************************************************************************************)
	T_Auto: 				BOOL;
	T_Manual:			BOOL;
	T_DryRun: 			BOOL;
	T_OriginSearch:		BOOL;
	T_Start:				BOOL;
	T_Stop:				BOOL;
	T_Reset :			BOOL;
 	T_Station_BypassP: 	ARRAY [0..50] OF BOOL;
	T_BypassDoor: 		BOOL;
	T_BypassBuzzer:		BOOL;
	T_BuzzerOff :			BOOL;
	T_AutoMsgAlarm: 		BOOL;
	T_StatusString: 		STRING;
	V_AutorunString: 		STRING;
(*************************************************************************************************************************************)
(*Auto*)
(*************************************************************************************************************************************)
	AutoPBMem: BOOL;
	NotAutoRunning:BOOL;

	pls_OriginSchRun: R_TRIG;
	OriginSchRunPls: BOOL;

(*************************************************************************************************************************************)
(*Manual*)
(*************************************************************************************************************************************)
	Pls_StepFwd: 	R_TRIG;
	Pls_StepBwd: 	R_TRIG;
	CycleTimer: 		TON;
	ManualCond: 		BOOL;
(*************************************************************************************************************************************)
	(* Error Handling*)
(*************************************************************************************************************************************)

	tmrEmgOn: TON;
	EmgPBTON :BOOL;

	tmrEmgOn_Air: TON;
	EmgPBTON_Air: BOOL;

	Reset:BOOL;
	pls_Reset :R_TRIG;
	ResetPls:BOOL;

	tmrDoorSwitch: TON;
	DoorSwTOFF: BOOL;

	tmrCurtainCrossed: TON;
	CurtainCrossedTON:BOOL;


END_VAR
(**************************************************************************************************************)
(* Auto Mode Selection*)
(**************************************************************************************************************)
IF T_Auto THEN
	AutoPBMem := TRUE;
END_IF;

IF( AutoPBMem OR MC.AutoRunning) AND NOT MC.Trouble THEN
	MC.AutoMode := TRUE;
ELSE
	MC.AutoMode := FALSE;
	AutoPBMem := FALSE;
END_IF;


(**************************************************************************************************************)
(*Manual Mode Selection*)
(**************************************************************************************************************)
IF T_Manual THEN
	AutoPBMem := FALSE;
END_IF;

IF NOT (AutoPBMem OR MC.AutoRunning OR MC.Trouble) THEN
	MC.ManualMode :=TRUE;
ELSE
	MC.ManualMode :=FALSE;
END_IF;


(**************************************************************************************************************)
(* Manual Interlocking *)
(**************************************************************************************************************)

ManualSafetyOK 	:=TRUE;
ManualCond 		:= MC.ManualMode AND ManualSafetyOK AND NOT mc.OriginSchRun;

(**************************************************************************************************************)
(* Manual General*)
(**************************************************************************************************************)

Pls_StepFwd(CLK:= I_StepFwdPB OR T_StepFwd);
M_StepFwdPls := Pls_StepFwd.Q;

Pls_StepBwd(CLK:= I_StepBwdPB OR T_StepBwd);
M_StepBwdPls := Pls_StepBwd.Q;


(**************************************************************************************************************)
(* Manual Stepping Mode*)
(**************************************************************************************************************)
IF (NOT T_StepStop) AND ManualCond THEN
	IF T_StepRun THEN
		M_StepRun := TRUE;
	END_IF;
ELSE
		M_StepRun := FALSE;
END_IF;


(* Display Status on Visio*)
T_StationError 		:= sc[T_Curr_Step_Station].MajorFault OR sc[T_Curr_Step_Station].MinorFault;
T_Origin 				:=sc[T_Curr_Step_Station].Origin;
V_StepRunCurrStation 	:= sc[T_Curr_Step_Station].Name;
V_StepRunStatus 		:= sc[T_Curr_Step_Station].Status;


FOR Loop := 1 TO Number_of_Station BY 1 DO
SC[Loop].M_Step		:= FALSE;
END_FOR

IF M_StepRun THEN
SC[T_Curr_Step_Station].M_Step	:= TRUE;
END_IF;


(* CycleTime Calculation*)
CycleTimer(IN:=M_StepRun , PT:=t#1100h , Q=> , ET=> );

IF M_StepRun THEN
T_ManualCycleTime :=CycleTimer.ET;
END_IF


(**************************************************************************************************************)
(*Reset Auto and Origin Bit*)
(**************************************************************************************************************)
	FOR LoopStation := 0 TO 20 BY 1 DO
		IF NOT (SC[LoopStation].AutoRun OR SC[LoopStation].M_Step OR MC.AutoMode)  THEN
			FOR Loop := 1 TO 10 BY 1 DO
				AutoDWord[LoopStation,Loop] :=0;
			END_FOR
		END_IF
	END_FOR

	FOR LoopStation := 0 TO 20 BY 1 DO
		IF NOT MC.OriginSchRun THEN
			FOR Loop := 1 TO 10 BY 1 DO
				OriginDWord[LoopStation,Loop] :=0;
			END_FOR
		END_IF
	END_FOR

(**************************************************************************************************************)
(*Origin Search Run*)
(**************************************************************************************************************)
IF MC.ManualMode AND NOT MC.AllOrigin AND NOT (MC.StationStopErr OR MC.Trouble OR MC.StopPressed )  THEN
	IF T_OriginSearch THEN
		MC.OriginSchRun  := TRUE;
	END_IF;
ELSE
	MC.OriginSchRun := FALSE;
END_IF;

pls_OriginSchRun(CLK:= MC.OriginSchRun);
OriginSchRunPls := pls_OriginSchRun.Q;


(**************************************************************************************************************)
(*Dry Run Mode Selection*)
(**************************************************************************************************************)
IF NOT MC.AutoRunning AND T_DryRun THEN
	MC.DryRun := TRUE;
END_IF;

IF NOT MC.AutoRunning AND NOT T_DryRun THEN
	MC.DryRun := FALSE;
	T_EndProd := FALSE;
END_IF;


(**************************************************************************************************************)
(* Machine Start *)
(**************************************************************************************************************)
IF MC.AutoMode AND NOT MC.Stop THEN
	IF (In_Start_PB OR T_Start) AND
		NOT MC.StationStopErr AND In_Start_Enable THEN
		MC.AutoRunning := TRUE;
	END_IF;
ELSE
	MC.AutoRunning := FALSE;
END_IF;

NotAutoRunning := NOT MC.AutoRunning;

IF MC.AutoRunning THEN
	V_AutorunString := 'Running';
ELSE
	V_AutorunString := 'Auto Mode';
END_IF


(**************************************************************************************************************)
(* Machine Stop *)
(**************************************************************************************************************)
IF MC.AutoRunning THEN
	IF NOT In_Stop_PB OR T_Stop OR In_EndProdWPCleared OR MC.StationStopErr THEN
		MC.StopPressed := TRUE;
	END_IF;
ELSE
	MC.StopPressed := FALSE;
END_IF;

IF MC.StopPressed AND AllStationStop THEN
	MC.Stop:=TRUE;
ELSE
	MC.Stop :=FALSE;
END_IF;


(**************************************************************************************************************)
(* Machine Status *)
(*From Station Status*)
(**************************************************************************************************************)

FOR Loop := 0 TO Number_of_Station BY 1  DO
IF NOT SC[Loop].Running THEN
AllStationStop := TRUE;
ELSE
AllStationStop := FALSE;
EXIT;
END_IF
END_FOR

FOR Loop := 0 TO Number_of_Station BY 1  DO
IF SC[Loop].Rdy THEN
MC.AllStationRdy := TRUE;
ELSE
MC.AllStationRdy := FALSE;
EXIT;
END_IF
END_FOR


FOR Loop := 0 TO Number_of_Station BY 1  DO
IF SC[Loop].NoWP THEN
MC.AllStationNoWP := TRUE;
ELSE
MC.AllStationNoWP := FALSE;
EXIT;
END_IF
END_FOR


FOR Loop := 0 TO Number_of_Station BY 1  DO
IF SC[Loop].Origin THEN
MC.AllOrigin:= TRUE;
ELSE
MC.AllOrigin := FALSE;
EXIT;
END_IF
END_FOR


(*Major Error for Immediate Stop*)
MC.Trouble:=E_EmgStop OR E_AirLow OR E_LightCurtain ;


FOR Loop := 0 TO Number_of_Station BY 1  DO
IF SC[Loop].MajorFault THEN
MC.Trouble:= TRUE;
END_IF
END_FOR

(*Minor Error for Stop after one cycle*)
MC.StationStopErr := E_SafetyDoorOpen  OR E_LightCurtain;

FOR Loop := 0 TO Number_of_Station BY 1  DO
IF SC[Loop].MinorFault THEN
MC.StationStopErr:= TRUE;
END_IF
END_FOR

(**************************************************************************************************************)
(* Auto Msg Alarm Display  *)
(**************************************************************************************************************)

IF MC.Trouble THEN
	T_StatusString := 'Machine Major Error';
ELSIF MC.StationStopErr THEN
	T_StatusString := 'Machine Station Error';
ELSIF MC.AutoMode THEN
	T_StatusString := 'Auto Mode';
ELSIF MC.ManualMode THEN
	T_StatusString := 'Manual Mode';
ELSIF MC.AutoRunning THEN
	T_StatusString := 'Auto Running';
END_IF

(**************************************************************************************************************)
(* For programmer Station Bypass - Debug Only*)
(**************************************************************************************************************)
IF NOT  MC.AutoRunning THEN

FOR Loop := 0 TO 20 DO
	IF T_Station_BypassP[Loop] THEN
            SC[Loop].Bypass := TRUE;
	ELSE
	    SC[Loop].Bypass := FALSE;
      END_IF;
END_FOR

END_IF;


(*************************************************************************************************************************************)
(* Reset Error And Warning Memory*)
(*************************************************************************************************************************************)

tmrEmgOn (IN := In_EmgOK, pt := T#1s);
EmgPBTON := tmrEmgOn.Q;

tmrEmgOn_Air (IN := In_EmgOK, pt := T#3s);
EmgPBTON_Air := tmrEmgOn_Air.Q;

Reset := T_Reset OR In_Reset_PB;

pls_Reset (CLK := Reset);
ResetPls := pls_Reset.Q;

(* Reset Error*)
	IF ResetPls AND EmgPBTON THEN
	FOR LoopStation := 0 TO 20 BY 1 DO
		FOR Loop := 1 TO 10 BY 1 DO
			ErrorDWord[LoopStation,Loop] :=0;
			WarningDWord[LoopStation,Loop] :=0;
		END_FOR
	END_FOR

			E_EmgStop:=FALSE;
			E_LightCurtain:=FALSE;
			E_AirLow :=FALSE;
			E_SafetyDoorOpen:=FALSE;

	END_IF;

(* Set Warning*)
MC.Warning := FALSE;
FOR LoopStation := 0 TO 20 BY 1 DO
	FOR Loop := 1 TO 10 DO
		IF WarningDWord[LoopStation,Loop]>0  THEN
			MC.Warning := TRUE;
		END_IF;
	END_FOR
END_FOR

T_AutoMsgAlarm := MC.Trouble OR MC.StationStopErr OR (NOT MC.AutoRunning AND NOT MC.AllOrigin) ;
(*************************************************************************************************************************************)
(*Error And Warning Summaries*)
(*************************************************************************************************************************************)
MC.ErrDetection := MC.AutoRunning OR MC.OriginSchRun;

(*************************************************************************************************************************************)
(*General Error and Trouble*)
(*************************************************************************************************************************************)

(*E-stop Error*)
IF NOT EmgPBTON THEN
	E_EmgStop := TRUE;
END_IF;

(*Safety Door Error*)
tmrDoorSwitch (in:= NOT In_Door_Sw, PT:= t#0.2S);
DoorSwTOFF := tmrDoorSwitch.Q;

IF  DoorSwTOFF AND NOT T_BypassDoor THEN
	E_SafetyDoorOpen := TRUE;
END_IF;

(*Air Low Error*)
IF EmgPBTON_Air AND NOT In_Pressure_Sw THEN
	E_AirLow := TRUE;
END_IF;

(*Light Curtain Crossed Error*)
tmrCurtainCrossed(IN := NOT In_LightCurtainOK, PT:= t#0.1s);
CurtainCrossedTON := tmrCurtainCrossed.Q;

IF NOT In_LightCurtainSafeToCross  AND NOT In_LightCurtainOK THEN
	E_LightCurtain := TRUE;
END_IF;

(**************************************************************************************************************)
(* General Output*)
(**************************************************************************************************************)

Out_RedTower := MC.Trouble OR ( MC.StationStopErr AND ON_1s);

Out_YelTower :=  MC.ManualMode OR ( MC.Warning AND ON_1s AND NOT  MC.Trouble AND NOT  MC.StationStopErr );

Out_GrnTower := (MC.AutoRunning AND NOT MC.StopPressed) OR (MC.StopPressed AND ON_1s) OR (MC.AutoMode AND ON_1s);

IF NOT (Out_RedTower OR MC.Warning) THEN
	T_BuzzerOff := FALSE;
END_IF

Out_Buzzer := (Out_RedTower OR (MC.Warning AND ON_1s)) AND NOT T_BuzzerOff AND NOT T_BypassBuzzer;
END_FUNCTION_BLOCK

(* POU Std_OnOffDev_Ctrl, LD *)
FUNCTION_BLOCK Std_OnOffDev_Ctrl

VAR_INPUT
	IN:BOOL;
	IN_DevName:STRING;
	In_Enable:BOOL;
	In_Reset:BOOL;


	(*Trigger*)
	In_AutoON:BOOL;
	In_OrgON:BOOL;

	(*Mechanical Interlock*)
	In_OnXLock:BOOL;

	(*Sensors*)
	In_ONSig:BOOL;

	(*Timer*)
	In_OnTON:TIME;
	in_Timeout:TIME;

END_VAR

VAR_OUTPUT
	Q:BOOL;
	Out_OnSV:BOOL;
	E_OnErr:BOOL;
	S_OnSig:BOOL;

END_VAR

VAR
	(* Trigger*)
	T_ManOn:BOOL;
	T_ManOff:BOOL;

	Loc_On:BOOL;
	On_TOut: TON;
	On_TON: TON;
	Loc_OnPls: BOOL;
	OnPls: R_TRIG;
	Out_RSErr:BOOL;
	OnPosPls: F_TRIG;

END_VAR
VAR_IN_OUT

END_VAR
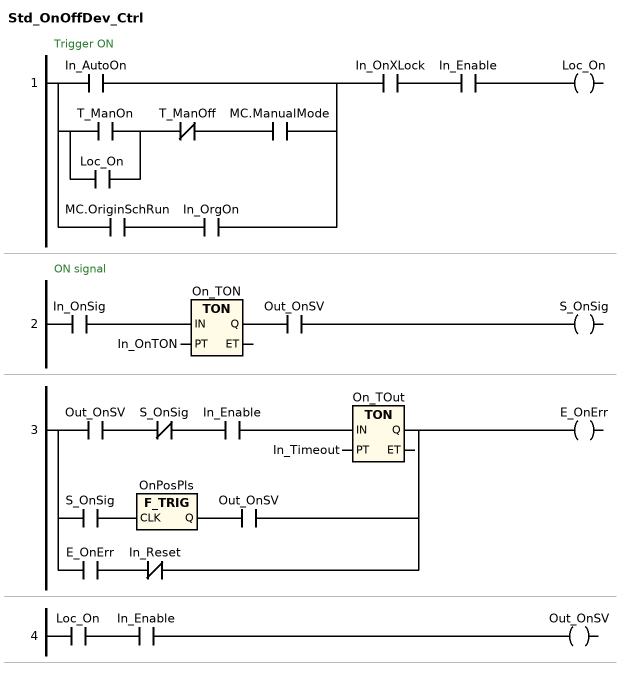
_LD_ (* Ladder Diagram *)
NETWORK 1 (* Trigger ON *)
	{ [In_AutoOn] | { [T_ManOn] | [Loc_On] } - [/T_ManOff] - [MC.ManualMode] | [MC.OriginSchRun] - [In_OrgOn] } - [In_OnXLock] - [In_Enable] --- (Loc_On)
NETWORK 2 (* ON signal *)
	[In_OnSig] - On_TON:TON(IN: *, PT: In_OnTON) - [Out_OnSV] --- (S_OnSig)
NETWORK 3
	{ [Out_OnSV] - [/S_OnSig] - [In_Enable] - On_TOut:TON(IN: *, PT: In_Timeout) | [S_OnSig] - OnPosPls:F_TRIG(CLK: *) - [Out_OnSV] | [E_OnErr] - [/In_Reset] } --- (E_OnErr)
NETWORK 4
	[Loc_On] - [In_Enable] --- (Out_OnSV)
_END_LD_
(* the same logic as Structured Text *)
(* Network 1: Trigger ON *)
Loc_On := (In_AutoOn OR (T_ManOn OR Loc_On) AND NOT T_ManOff AND MC.ManualMode OR MC.OriginSchRun AND In_OrgOn) AND In_OnXLock AND In_Enable;
(* Network 2: ON signal *)
On_TON(IN := In_OnSig, PT := In_OnTON);
S_OnSig := On_TON.Q AND Out_OnSV;
(* Network 3 *)
On_TOut(IN := Out_OnSV AND NOT S_OnSig AND In_Enable, PT := In_Timeout);
OnPosPls(CLK := S_OnSig);
E_OnErr := On_TOut.Q OR OnPosPls.Q AND Out_OnSV OR E_OnErr AND NOT In_Reset;
(* Network 4 *)
Out_OnSV := Loc_On AND In_Enable;
END_FUNCTION_BLOCK

(* POU Std_Password_Ctrl, ST *)
(* @OBJECTFLAGS := '0, 8' *)
FUNCTION_BLOCK Std_Password_Ctrl
VAR_INPUT
	In_PasswordConfig:STRING;
	In_SelectedPasswordLvl:INT; (* 0   - operator, 1 - Supervisor, 3-Maintenance *)
END_VAR
VAR_OUTPUT

END_VAR
VAR RETAIN
	In_EntryPasswordString:STRING;
	In_NewPasswordString1:STRING;
	In_NewPasswordString2:STRING;
	In_CurrPasswordStringOperator:STRING;
	In_CurrPasswordStringSupervisor:STRING;
	In_CurrPasswordStringMaintenance:STRING;
	In_EnterPassword:BOOL;
	In_ChangePassword:BOOL;

	Out_PasswordOK:BOOL;
	Out_PasswordChanged:BOOL;
	Out_CurrPasswordString:STRING;
	Out_StatusString:STRING;
	Out_PasswordConfig:BOOL;
	Out_CurrentPasswordLvl:INT; (* 0   - operator, 1 - Supervisor, 3-Maintenance *)

	PasswordOK:BOOL;
	tmrStatusChanged: TON;
	StatusChanged: BOOL;
	StatusChangedTON: BOOL;

	PaswordEnteredPls:BOOL;
	pls_PasswordEntered:R_TRIG;
	NewPaswordEnteredPls:BOOL;
	pls_NewPasswordEntered:R_TRIG;

END_VAR
tmrStatusChanged(IN := StatusChanged, PT:= t#2s);
StatusChangedTON := tmrStatusChanged.Q;

pls_PasswordEntered(CLK:= In_EnterPassword);
PaswordEnteredPls := pls_PasswordEntered.Q;

pls_NewPasswordEntered(CLK:= In_ChangePassword);
NewPaswordEnteredPls := pls_NewPasswordEntered.Q;

IF StatusChangedTON THEN
	Out_StatusString := '';
	StatusChanged := FALSE;
END_IF

(************************************************************************************************)
(* Password Entry*)
(************************************************************************************************)

IF PaswordEnteredPls THEN
	IF (In_EntryPasswordString =In_CurrPasswordStringOperator AND In_SelectedPasswordLvl =0) OR
	(In_EntryPasswordString =In_CurrPasswordStringSupervisor AND In_SelectedPasswordLvl =1) OR
	(In_EntryPasswordString =In_CurrPasswordStringMaintenance AND In_SelectedPasswordLvl =2)  THEN
		Out_PasswordOK := TRUE;
		PasswordOK := TRUE;
		Out_PasswordConfig := FALSE;
		Out_StatusString := 'Password OK!';
		Out_CurrentPasswordLvl:=In_SelectedPasswordLvl;
	ELSIF In_EntryPasswordString = In_PasswordConfig THEN
		Out_PasswordOK := TRUE;
		Out_PasswordConfig := TRUE;
		PasswordOK := TRUE;
		Out_StatusString := 'Password Config OK!';
	ELSE
		Out_PasswordConfig := FALSE;
		Out_StatusString := 'Wrong Password!';
	END_IF
	StatusChanged := TRUE;
ELSE
	Out_PasswordOK := FALSE;
END_IF



(************************************************************************************************)
(* Password Change*)
(************************************************************************************************)

IF NewPaswordEnteredPls  THEN
	IF( In_EntryPasswordString = In_CurrPasswordStringMaintenance) OR In_SelectedPasswordLvl < 2 THEN
		IF In_NewPasswordString1 <> '' AND In_NewPasswordString2 <>''  THEN
			IF In_NewPasswordString1 = In_NewPasswordString2 THEN
					CASE In_SelectedPasswordLvl OF
						0: In_CurrPasswordStringOperator :=In_NewPasswordString1;
						1: In_CurrPasswordStringSupervisor :=In_NewPasswordString1;
						2: In_CurrPasswordStringMaintenance :=In_NewPasswordString1;
					END_CASE
				Out_PasswordChanged := TRUE;
				Out_StatusString := 'Password Changed!';
			ELSE
				Out_StatusString := 'New Passwords not match!';
			END_IF
		ELSE
			Out_StatusString := 'New Password is empty!';
		END_IF
	ELSE
		Out_StatusString := 'Old Password is wrong!';
	END_IF
	StatusChanged := TRUE;
ELSE
	Out_PasswordChanged := FALSE;
END_IF

(* Reset password String *)
IF PaswordEnteredPls OR NewPaswordEnteredPls THEN
	In_EntryPasswordString :='';
	In_NewPasswordString1:='';
	In_NewPasswordString2:='';
END_IF
END_FUNCTION_BLOCK

(* POU Std_StepCase, ST *)
FUNCTION_BLOCK Std_StepCase

VAR_INPUT
	IN:BOOL;
	Step_Number: INT;
END_VAR
VAR_OUTPUT
	Q: BOOL;
	Step: ARRAY [0..9999] OF BOOL;
END_VAR

VAR
	Loop: INT;
END_VAR
FOR  Loop := 0 TO 9999 DO

IF Step_Number = Loop  THEN
Step[Loop] :=TRUE;
ELSE
Step[Loop] := FALSE;
END_IF

END_FOR
END_FUNCTION_BLOCK

(* Visualisation Blue_Ind
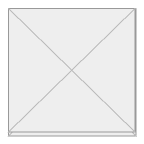
bitmap at (0,0)-(128,128): c:\flexlink\bitmap\button_blank_blue_01.bmp
bitmap at (0,0)-(127,124): c:\flexlink\bitmap\\button_blank_gray_01.bmp
*)

(* Visualisation ButtonGreenInd
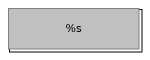
rectangle at (0,0)-(131,41): text "%s"; shows $Text$; alarm colour if $ColourTag$; taps $TapTag$; runs INTERN ASSIGN $ValueTag$:=($AssignValue$)
1 more shapes without text or variables
*)

(* Visualisation Green_Ind
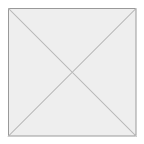
bitmap at (0,0)-(128,128): c:\flexlink\bitmap\button_blank_gray_01.bmp
bitmap at (0,0)-(128,128): c:\flexlink\bitmap\button_blank_green_01.bmp
*)

(* Visualisation Indradrive
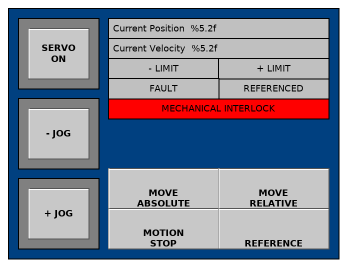
rounded rectangle at (10,170)-(91,241): alarm colour if $Inst$.In_JogFwd
rounded rectangle at (10,90)-(91,161): alarm colour if $Inst$.In_JogBwd
rounded rectangle at (10,10)-(91,81): alarm colour if $Inst$.In_ServoOn
button at (20,20)-(81,71): text "SERVO / ON"; toggles $Inst$.In_ServoOn
button at (20,100)-(81,151): text "- JOG"; taps $Inst$.In_JogBwd
button at (20,180)-(81,231): text "+ JOG"; taps $Inst$.In_JogFwd
rounded rectangle at (100,90)-(321,111): text "MECHANICAL INTERLOCK"; invisible if $Inst$.In_MoveXLock
rectangle at (100,10)-(321,31): text "Current Position  %5.2f"; shows $Inst$.Out_CurrPos
rectangle at (100,30)-(321,51): text "Current Velocity  %5.2f"; shows $Inst$.Out_CurrVel
rounded rectangle at (210,70)-(321,91): text "REFERENCED"; alarm colour if $Inst$.Out_Referenced
rounded rectangle at (100,50)-(211,71): text "- LIMIT"; alarm colour if $Inst$.Out_PosLimit
rounded rectangle at (210,50)-(321,71): text "+ LIMIT"; alarm colour if $Inst$.Out_PosLimit
button at (100,160)-(211,201): text "MOVE / ABSOLUTE"; taps $Inst$.In_MoveAbs
button at (210,160)-(321,201): text "MOVE / RELATIVE"; taps $Inst$.In_MoveRel
button at (100,200)-(211,241): text "MOTION / STOP"; taps $Inst$.In_StopMove
button at (210,200)-(321,241): text "REFERENCE"; taps $Inst$.In_MoveHome
rounded rectangle at (100,70)-(211,91): text "FAULT"; alarm colour if $Inst$.Out_Error
1 more shapes without text or variables
2 elements of other kinds (tables, trends, ...) not read
*)

(* Visualisation IO_Monitor
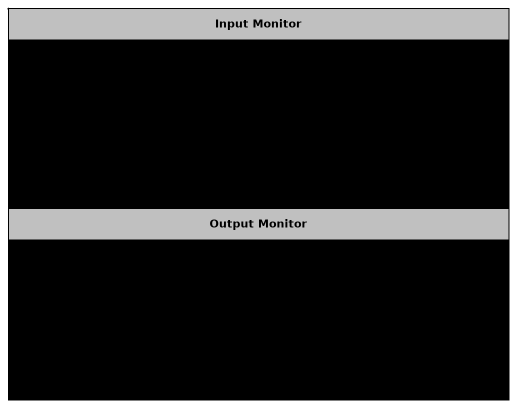
rectangle at (0,0)-(0,0): alarm colour if InputByte[INDEX].7
rectangle at (0,0)-(0,0): alarm colour if InputByte[INDEX].6
rectangle at (0,0)-(0,0): alarm colour if InputByte[INDEX].5
rectangle at (0,0)-(0,0): alarm colour if InputByte[INDEX].4
rectangle at (0,0)-(0,0): alarm colour if InputByte[INDEX].3
rectangle at (0,0)-(0,0): alarm colour if InputByte[INDEX].2
rectangle at (0,0)-(0,0): alarm colour if InputByte[INDEX].1
rectangle at (0,0)-(0,0): alarm colour if InputByte[INDEX].0
rectangle at (0,0)-(501,32): text "Input Monitor"
rectangle at (0,0)-(0,0): alarm colour if OutputByte[INDEX].7
rectangle at (0,0)-(0,0): alarm colour if OutputByte[INDEX].6
rectangle at (0,0)-(0,0): alarm colour if OutputByte[INDEX].5
rectangle at (0,0)-(0,0): alarm colour if OutputByte[INDEX].4
rectangle at (0,0)-(0,0): alarm colour if OutputByte[INDEX].3
rectangle at (0,0)-(0,0): alarm colour if OutputByte[INDEX].2
rectangle at (0,0)-(0,0): alarm colour if OutputByte[INDEX].1
rectangle at (0,0)-(0,0): alarm colour if OutputByte[INDEX].0
rectangle at (0,200)-(501,232): text "Output Monitor"
1 more shapes without text or variables
*)

(* Visualisation MANUAL_STEP
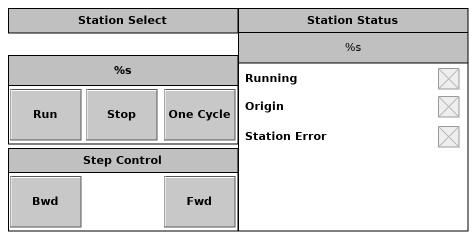
rectangle at (0,47)-(230,78): text "%s"; shows .V_StepRunCurrStation
rounded rectangle at (20,-3)-(209,28): text "Station Select"
button at (2,81)-(73,132): text "Run"; taps .T_StepRun
button at (78,81)-(149,132): text "Stop"; taps .T_StepStop
button at (156,81)-(227,132): text "One Cycle"; toggles .T_OneCycleRun
rounded rectangle at (20,137)-(209,168): text "Step Control"
button at (2,168)-(73,219): text "Bwd"; taps .T_StepBwd
button at (156,168)-(227,219): text "Fwd"; taps .T_StepFwd
rounded rectangle at (250,-3)-(439,28): text "Station Status"
rounded rectangle at (235,55)-(331,86): text "Running"
rounded rectangle at (235,83)-(331,114): text "Origin"
rounded rectangle at (235,113)-(331,144): text "Station Error"
rectangle at (230,24)-(460,55): text "%s"; shows V_StepRunStatus
embedded screen at (430,118)-(451,139): Red_Ind
embedded screen at (430,88)-(451,109): Green_Ind
embedded screen at (430,60)-(451,81): Green_Ind
6 more shapes without text or variables
1 elements of other kinds (tables, trends, ...) not read
*)

(* Visualisation Red_Ind
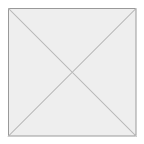
bitmap at (0,0)-(128,128): c:\flexlink\bitmap\button_blank_gray_01.bmp
bitmap at (0,0)-(128,128): c:\flexlink\bitmap\button_blank_red_01.bmp
*)

(* Visualisation Std_Alm_Ctrl_Button
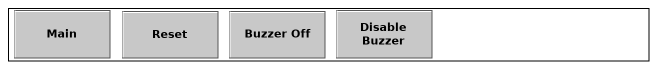
button at (6,1)-(102,49): text "Main"; opens TP00_MAIN
button at (114,2)-(210,49): text "Reset"; taps $Inst$.T_Reset
rectangle at (229,2)-(310,48): text "Buzzer Off"; alarm colour if .T_BuzzerOff; toggles $Inst$.T_BuzzerOff
rectangle at (330,4)-(421,46): text "Disable / Buzzer"; alarm colour if .T_BypassBuzzer; toggles $Inst$.T_BypassBuzzer
3 more shapes without text or variables
*)

(* Visualisation Std_Cylinder_Ctrl
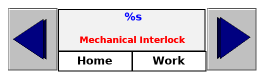
rounded rectangle at (48,0)-(195,42): text "%s"; shows $Inst$.IN_CylName
rounded rectangle at (48,42)-(122,62): text "Home"; invisible if $Inst$.E_HomeErr; alarm colour if $Inst$.S_HomePos
rounded rectangle at (122,42)-(196,62): text "Work"; invisible if $Inst$.E_WorkErr; alarm colour if $Inst$.S_WorkPos
group at (-2,-1)-(47,61)
  button at (0,0)-(49,62): taps $Inst$.In_ManHome
group at (197,-1)-(246,61)
  button at (0,0)-(49,61): taps $Inst$.In_ManWork
rounded rectangle at (49,21)-(196,41): text "Mechanical Interlock"; invisible if NOT (NOT $Inst$.In_WorkXLock AND $Inst$.T_ManWork)
rounded rectangle at (49,21)-(196,41): text "Mechanical Interlock"; invisible if NOT (NOT $Inst$.In_HomeXLock AND $Inst$.T_ManHome)
rounded rectangle at (48,42)-(122,62): text "Home"; invisible if NOT $Inst$.E_HomeErr; alarm colour if $Inst$.E_HomeErr
rounded rectangle at (122,42)-(196,62): text "Work"; invisible if NOT $Inst$.E_WorkErr; alarm colour if $Inst$.E_WorkErr
4 more shapes without text or variables
*)

(* Visualisation Std_IAI_16Point
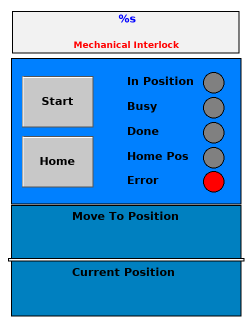
rounded rectangle at (117,58)-(193,89): text "In Position"
ellipse at (195,64)-(216,85): alarm colour if $Inst$.S_InPos
rounded rectangle at (117,83)-(193,114): text "Busy"
ellipse at (195,89)-(216,110): alarm colour if NOT $Inst$.In_PEND
rounded rectangle at (117,108)-(193,139): text "Done"
ellipse at (195,114)-(216,135): alarm colour if $Inst$.In_PEND
rounded rectangle at (117,133)-(193,164): text "Home Pos"
ellipse at (195,139)-(216,160): alarm colour if $Inst$.S_InHome
rounded rectangle at (117,157)-(193,188): text "Error"
ellipse at (195,163)-(216,184): alarm colour if .E4_Scan_IAI_Alm OR .E4_Scan_IAI_MovPos OR .E4_Scan_IAI_PosAlm
button at (14,68)-(85,119): text "Start"; taps $Inst$.T_ManStart
button at (14,128)-(85,179): text "Home"; taps $Inst$.T_ManHome
rounded rectangle at (62,193)-(175,224): text "Move To Position"
rounded rectangle at (62,249)-(175,280): text "Current Position"
rounded rectangle at (4,3)-(231,45): text "%s"; shows $Inst$.IN_Name
rounded rectangle at (45,27)-(192,47): text "Mechanical Interlock"; invisible if NOT (NOT $Inst$.In_Mec_Interlock AND ($Inst$.In_ManStart OR $Inst$.In_ManHome))
4 more shapes without text or variables
2 elements of other kinds (tables, trends, ...) not read
*)

(* Visualisation Std_IV_Vision_Ctrl
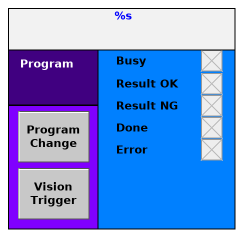
button at (10,103)-(81,154): text "Program / Change"; taps $Inst$.T_ManualTrigger
rounded rectangle at (106,42)-(182,63): text "Busy"
rounded rectangle at (106,65)-(182,86): text "Result OK"
rounded rectangle at (106,109)-(182,130): text "Done"
rounded rectangle at (106,131)-(182,152): text "Error"
rounded rectangle at (106,87)-(182,108): text "Result NG"
embedded screen at (193,42)-(214,63): Green_Ind
embedded screen at (193,65)-(214,86): Green_Ind
embedded screen at (193,87)-(214,108): Red_Ind
embedded screen at (193,109)-(214,130): Green_Ind
embedded screen at (193,131)-(214,152): Red_Ind
rounded rectangle at (10,40)-(97,71): text "Program"
rounded rectangle at (0,0)-(227,42): text "%s"; shows $Inst$.IN_Name$Num$
button at (10,160)-(81,211): text "Vision / Trigger"; taps $Inst$.T_ManualTrigger
3 more shapes without text or variables
1 elements of other kinds (tables, trends, ...) not read
*)

(* Visualisation Std_Main_Ctrl_Button
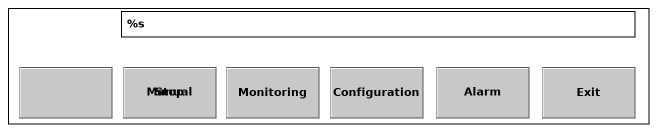
rectangle at (11,-1)-(142,30): text "Machine Status:"
rectangle at (113,1)-(627,27): text "%s"; shows $Inst$.T_StatusString; alarm colour if $Inst$.T_AutoMsgAlarm
button at (218,57)-(311,108): text "Monitoring"; opens TP50_Monitoring; dynamic style cmd_ManMode
button at (322,57)-(415,108): text "Configuration"; invisible if $Inst$.InOut_SC.AutoRunning; opens TP30_PASSWORD; dynamic style cmd_ManMode
button at (428,57)-(521,108): dynamic style cmd_ManMode
button at (534,57)-(627,108): text "Exit"; invisible if $Inst$.InOut_SC.AutoRunning; opens TP00_MAIN_EXIT; runs INTERN EXITPROGRAM; dynamic style cmd_ManMode
rectangle at (432,59)-(517,105): text "Alarm"; alarm colour if $Inst$.Out_RedTower; opens TP80_ALARM
button at (115,57)-(208,108): dynamic style cmd_ManMode
rectangle at (119,59)-(204,105): text "Manual"; invisible if MC.AutoRunning; alarm colour if MC.ManualMode; taps $Inst$.T_Manual; opens TP10_MANUAL
rectangle at (119,59)-(204,105): text "Stop"; invisible if NOT MC.AutoRunning; alarm colour if MC.StopPressed AND On_1s; taps $Inst$.T_Stop
button at (11,57)-(104,108): dynamic style btn_Auto
1 more shapes without text or variables
3 elements of other kinds (tables, trends, ...) not read
*)

(* Visualisation Std_NewPassWord
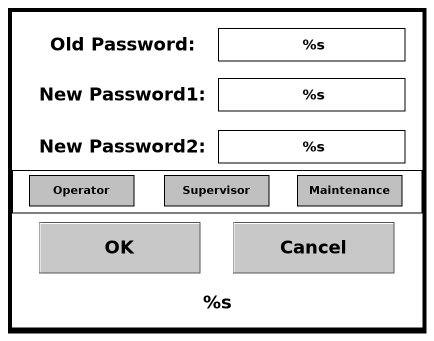
rounded rectangle at (17,20)-(206,51): text "Old Password:"; invisible if In_SelectedPasswordLvl < 2
rectangle at (207,19)-(394,52): text "%s"; shows .Password_Control.In_EntryPasswordString; invisible if In_SelectedPasswordLvl < 2; editable 0..10
button at (28,213)-(189,264): text "OK"; taps .Password_Control.In_ChangePassword
button at (222,213)-(383,264): text "Cancel"; opens TP40_SETTING
rounded rectangle at (9,278)-(404,309): text "%s"; shows .Password_Control.Out_StatusString
rounded rectangle at (17,70)-(206,101): text "New Password1:"
rectangle at (207,69)-(394,102): text "%s"; shows .Password_Control.In_NewPasswordString1; editable 0..10
rounded rectangle at (17,122)-(206,153): text "New Password2:"
rectangle at (207,121)-(394,154): text "%s"; shows .Password_Control.In_NewPasswordString2; editable 0..10
rounded rectangle at (18,166)-(123,197): text "Operator"; alarm colour if .Password_Control.In_SelectedPasswordLvl = 0; runs INTERN ASSIGN Password_Control.In_SelectedPasswordLvl:=(0)
rounded rectangle at (153,166)-(258,197): text "Supervisor"; alarm colour if .Password_Control.In_SelectedPasswordLvl = 1; runs INTERN ASSIGN Password_Control.In_SelectedPasswordLvl:=(1)
rounded rectangle at (286,166)-(391,197): text "Maintenance"; alarm colour if .Password_Control.In_SelectedPasswordLvl = 2; runs INTERN ASSIGN Password_Control.In_SelectedPasswordLvl:=(2)
3 more shapes without text or variables
3 elements of other kinds (tables, trends, ...) not read
*)

(* Visualisation Std_OnOffDev_Ctrl
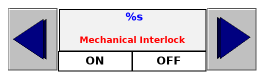
rounded rectangle at (50,0)-(197,42): text "%s"; shows $Inst$.IN_DevName
rounded rectangle at (49,42)-(123,62): text "ON"; alarm colour if $Inst$.S_OnSig
rounded rectangle at (123,42)-(197,62): text "OFF"; alarm colour if NOT $Inst$.S_OnSig
rounded rectangle at (50,21)-(197,41): text "Mechanical Interlock"; invisible if NOT (NOT $Inst$.In_OnXLock AND $Inst$.T_ManOn)
6 more shapes without text or variables
*)

(* Visualisation Std_Password
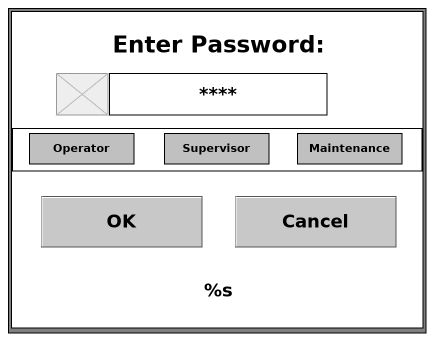
rounded rectangle at (89,20)-(330,51): text "Enter Password:"
rectangle at (100,64)-(318,106): text "****"; shows .Password_Control.In_EntryPasswordString; editable 0..10
button at (32,187)-(193,238): text "OK"; taps .Password_Control.In_EnterPassword
button at (226,187)-(387,238): text "Cancel"; opens TP00_MAIN
rounded rectangle at (89,266)-(330,297): text "%s"; shows .Password_Control.Out_StatusString
bitmap at (47,64)-(99,106): c:\flexlink\bitmap\lock.bmp
rounded rectangle at (20,124)-(125,155): text "Operator"; alarm colour if .Password_Control.In_SelectedPasswordLvl = 0; runs INTERN ASSIGN Password_Control.In_SelectedPasswordLvl:=(0)
rounded rectangle at (155,124)-(260,155): text "Supervisor"; alarm colour if .Password_Control.In_SelectedPasswordLvl = 1; runs INTERN ASSIGN Password_Control.In_SelectedPasswordLvl:=(1)
rounded rectangle at (288,124)-(393,155): text "Maintenance"; alarm colour if .Password_Control.In_SelectedPasswordLvl = 2; runs INTERN ASSIGN Password_Control.In_SelectedPasswordLvl:=(2)
3 more shapes without text or variables
3 elements of other kinds (tables, trends, ...) not read
*)

(* Visualisation Std_VacuumVal_Ctrl
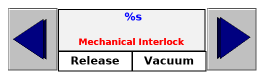
rounded rectangle at (48,0)-(195,42): text "%s"; shows $Inst$.IN_Name
rounded rectangle at (48,42)-(122,62): text "Release"; invisible if $Inst$.E_PurgeErr; alarm colour if $Inst$.S_Release
rounded rectangle at (122,42)-(196,62): text "Vacuum"; invisible if $Inst$.E_VacuumErr; alarm colour if $Inst$.S_Vacuum
group at (-2,-1)-(47,61)
  button at (0,0)-(49,62): taps $Inst$.In_ManHome
group at (197,-1)-(246,61)
  button at (0,0)-(49,61): taps $Inst$.In_ManWork
rounded rectangle at (48,23)-(195,43): text "Mechanical Interlock"; invisible if NOT (NOT $Inst$.In_VacuumX AND $Inst$.T_ManVacuum)
rounded rectangle at (48,23)-(195,43): text "Mechanical Interlock"; invisible if NOT (NOT $Inst$.In_PurgeX AND $Inst$.T_ManPurge)
rounded rectangle at (48,42)-(122,62): text "Release"; invisible if NOT $Inst$.E_PurgeErr; alarm colour if $Inst$.E_PurgeErr
rounded rectangle at (122,42)-(196,62): text "Vacuum"; invisible if NOT $Inst$.E_VacuumErr; alarm colour if $Inst$.E_VacuumErr
4 more shapes without text or variables
*)

(* Visualisation ToggleSwitch1
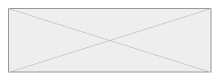
bitmap at (0,0)-(203,63): c:\flexlink\bitmap\toggleswitchgreen.bmp
bitmap at (0,0)-(203,64): c:\flexlink\bitmap\toggleswitchred.bmp
*)

(* Visualisation Yellow_Ind
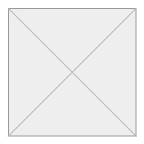
bitmap at (0,0)-(128,128): c:\flexlink\bitmap\button_blank_gray_01.bmp
bitmap at (0,0)-(128,128): c:\flexlink\bitmap\button_blank_yellow_01.bmp
*)
